FUNCTION_BLOCK EM_Filling IMPLEMENTS  ITF_EM_Filling
VAR_INPUT
END_VAR
VAR_OUTPUT
END_VAR
VAR
END_VAR

//voor het voorbeeld

END_FUNCTION_BLOCK

(* stored: Version 1.1.0.1, ProductVersion 3.1.4024.12
   POU EM_Filling: Id {e31cb704-0c01-44ce-bc30-5b4bfac97888}, SpecialFunc None *)
